Fanuc KAREL source: kt00254.KL

-- PROVISIONAL review KL for V940-1; original PC SHA256 7eb956accff21696571dc584c5fd7080844faed4c44c10b71a1c26902b7a4643
-- Incomplete behavior may be omitted. Consult companion uncertainty JSON. Do not deploy.
PROGRAM KT00254
%NOLOCKGROUP
VAR
  OUT : INTEGER
-- UNRESOLVED_DECL H1 type=002017
-- UNRESOLVED_DECL Y2 type=002018
BEGIN
  -- V9_ZERO_TABLE_METADATA_HINT layout=0001; no indexed target words; source/name/runtime held
  -- UNRESOLVED_PC offsets 5-19; opcodes 2E,22,9D,33,B4
  -- UNRESOLVED_PC offsets 24-38; opcodes 2E,22,9D,33,B2
  -- UNRESOLVED_PC offsets 43-68; opcodes 22,9D,33,B3,22,9D,33,B1,47,23
  -- UNRESOLVED_PC offsets 73-77; opcodes 7F
END KT00254
